{attribute addProperty BoxType "KL3351-0003"}
{attribute addProperty Id "StatusAT %I*USINT000Ud_RegInAT %I*INT000UrefAT %I*INT000CtrlAT %Q*USINT000RegOutAT %Q*INT000Ctrl1AT %Q*USINT000"}
{attribute addProperty CRC "2212893950"}
{attribute addProperty SizeInBites "0"}
{attribute addProperty SizeInBytes "0"}
TYPE Channel_83E614FE :
STRUCT
	{attribute addProperty Name "Status"}
	Status AT %I* : USINT;
	{attribute addProperty Name "Ud_RegIn"}
	Ud_RegIn AT %I* : INT;
	{attribute addProperty Name "Uref"}
	Uref AT %I* : INT;
	{attribute addProperty Name "Ctrl"}
	Ctrl AT %Q* : USINT;
	{attribute addProperty Name "RegOut"}
	RegOut AT %Q* : INT;
	{attribute addProperty Name "Ctrl1"}
	Ctrl1 AT %Q* : USINT;
END_STRUCT
END_TYPE

(* stored: Version 1.2.0.0, ProductVersion 3.1.4024.9
   DUT Channel_83E614FE: Id {845c95dc-e8e9-45f3-9026-95e7acf3ed19} *)
